// TwinCAT 3 PLC project _04_SingletonByProxy
// ProgramVersion: 3.1.4023.0
// libraries:
//   Tc2_Standard, * (Beckhoff Automation GmbH)
//   Tc2_System, * (Beckhoff Automation GmbH)
//   Tc3_Module, * (Beckhoff Automation GmbH)
// project tree:
//   / MAIN.TcPOU, PlcTask.TcTTO
//   Singleton Pattern/Abstraction/ I_Singleton.TcIO, MySingleton.TcPOU, Singleton.TcPOU
//   Singleton Pattern/ P_Singleton.TcPOU
//   Singleton Pattern/SingletonByProxy/ I_MessageLogger.TcIO, MessageLogger.TcPOU, MessageLoggerSingleton.TcPOU
// (motion and I/O tree: see PLC project 13_decorator)
// real-time tasks:
//   TASK PlcTask: cycle T#10ms, priority 20, ADS port 350
// variable links:

CONFIGURATION _04_SingletonByProxy
    RESOURCE PLC ON TwinCAT3
        TASK PlcTask(INTERVAL := T#10ms, PRIORITY := 20);
        PROGRAM MAIN WITH PlcTask : MAIN;
    END_RESOURCE
END_CONFIGURATION

// ---- Singleton Pattern/Abstraction/I_Singleton.TcIO
INTERFACE I_Singleton

METHOD Message : String
VAR_INPUT
END_VAR
END_METHOD

END_INTERFACE

// ---- Singleton Pattern/SingletonByProxy/I_MessageLogger.TcIO
INTERFACE I_MessageLogger

METHOD LogMessage : String
VAR_INPUT
	Message			: STRING;
END_VAR
END_METHOD

PROPERTY message : string
GET
END_GET
END_PROPERTY

END_INTERFACE

// ---- MAIN.TcPOU
PROGRAM MAIN
VAR
END_VAR

(* 
	GOF 		Ensure a class only has one instance, and provide a global point of access to it.
*)
P_Singleton();

END_PROGRAM

// ---- Singleton Pattern/P_Singleton.TcPOU
(*
	For now there seems not to be a possibility to create a real single singleton. 
	The only solution found is the one by proxy, but that also means extra work since methods have to be written in the proxy.
*)
PROGRAM P_Singleton
VAR
	messageLogger				: MessageLogger;
	messageLogger1				: MessageLogger;
	messageLogger2				: MessageLogger;
	myMessage					: STRING;
	myMessage1					: STRING := 'Message 1';
	myMessage2					: STRING := 'Message 2';
	myMessage3					: STRING := 'Message 3';
END_VAR

// Log 'message 1' to the first messagelogger instance
messageLogger.LogMessage(myMessage1);
myMessage := messageLogger.message;

// Log 'message 2' to a second messagelogger instance
messageLogger1.LogMessage(myMessage2);
myMessage := messageLogger.message;
myMessage := messageLogger1.message;

// Log 'message 3' to a third messagelogger instance
messageLogger2.LogMessage(myMessage3);
myMessage := messageLogger.message;
myMessage := messageLogger2.message;

END_PROGRAM

// ---- Singleton Pattern/SingletonByProxy/MessageLogger.TcPOU
{attribute 'no_explicit_call' := 'MySingleton is a CLASS and must be accessed using methods or properties'}
FUNCTION_BLOCK MessageLogger IMPLEMENTS I_MessageLogger
VAR_STAT 	// VAR_STAT makes sure all new instances use the same initialized vars
	messageLogger					: I_MessageLogger;				
	messageLoggerSingleton			: POINTER TO MessageLoggerSingleton;
END_VAR

METHOD FB_exit : BOOL
VAR_INPUT
	bInCopyCode : BOOL; // if TRUE, the exit method is called for exiting an instance that is copied afterwards (online change).
END_VAR
// Delete the dynamic instance at FB_exit 
IF messageLoggerSingleton <> 0	THEN
	messageLogger := 0;					// Clear interface
	__DELETE(messageLoggerSingleton);	// Delete the instance
	messageLoggerSingleton:=0;			// Clear the pointer
END_IF
END_METHOD

METHOD FB_init : BOOL
VAR_INPUT
	bInitRetains : BOOL; // if TRUE, the retain variables are initialized (warm start / cold start)
	bInCopyCode : BOOL;  // if TRUE, the instance afterwards gets moved into the copy code (online change)
END_VAR
// first instance? 
IF messageLoggerSingleton = 0	THEN
	messageLoggerSingleton := __NEW(messageLoggerSingleton);
	messageLogger := messageLoggerSingleton^;
END_IF
END_METHOD

METHOD LogMessage : STRING
VAR_INPUT
	message			: STRING;
END_VAR
IF messageLogger <> 0 THEN
	messageLogger.LogMessage(message);
END_IF
END_METHOD

{warning 'add property implementation'}
PROPERTY message : STRING
GET
message := messageLogger.message;
END_GET
END_PROPERTY

END_FUNCTION_BLOCK

// ---- Singleton Pattern/Abstraction/MySingleton.TcPOU
{attribute 'no_explicit_call' := 'MySingleton is a CLASS and must be accessed using methods or properties'}
FUNCTION_BLOCK MySingleton IMPLEMENTS I_Singleton
VAR 
	singleton					: I_Singleton;	// define the static class instance	
	singletonInstance			: POINTER TO Singleton;
END_VAR

METHOD FB_exit : BOOL
VAR_INPUT
	bInCopyCode : BOOL; // if TRUE, the exit method is called for exiting an instance that is copied afterwards (online change).
END_VAR
// first instance? 
IF singletonInstance <> 0	THEN
	singleton := 0;
	__DELETE(singletonInstance);
	singletonInstance:=0;
END_IF
END_METHOD

METHOD FB_init : BOOL
VAR_INPUT
	bInitRetains : BOOL; // if TRUE, the retain variables are initialized (warm start / cold start)
	bInCopyCode : BOOL;  // if TRUE, the instance afterwards gets moved into the copy code (online change)
END_VAR
// first instance? 
IF singletonInstance = 0	THEN
	singletonInstance := __NEW(Singleton);
	singleton := singletonInstance^;
END_IF
END_METHOD

METHOD FB_reinit : BOOL
VAR_INPUT
END_VAR
__DELETE(singletonInstance);
singleton := 0;
END_METHOD

METHOD Message : STRING
IF singleton <> 0 THEN
	Message := singleton.Message();
END_IF
END_METHOD

END_FUNCTION_BLOCK

// ---- Singleton Pattern/Abstraction/Singleton.TcPOU
{attribute 'enable_dynamic_creation'}
{attribute 'no_explicit_call' := 'Singleton is a CLASS and must be accessed using methods or properties'}
FUNCTION_BLOCK Singleton IMPLEMENTS I_Singleton

METHOD Message : STRING
Message := 'myMessage';
END_METHOD

END_FUNCTION_BLOCK

// ---- Singleton Pattern/SingletonByProxy/MessageLoggerSingleton.TcPOU
{attribute 'enable_dynamic_creation'}
{attribute 'no_explicit_call' := 'Singleton is a CLASS and must be accessed using methods or properties'}
FUNCTION_BLOCK MessageLoggerSingleton IMPLEMENTS I_MessageLogger // USE MessageLogger!!
VAR
	_message			: STRING;
END_VAR

METHOD LogMessage : STRING
VAR_INPUT
	message			: STRING;
END_VAR
_message := message;
END_METHOD

{warning 'add property implementation'}
PROPERTY message : STRING
GET
message  := _message;
END_GET
END_PROPERTY

END_FUNCTION_BLOCK
